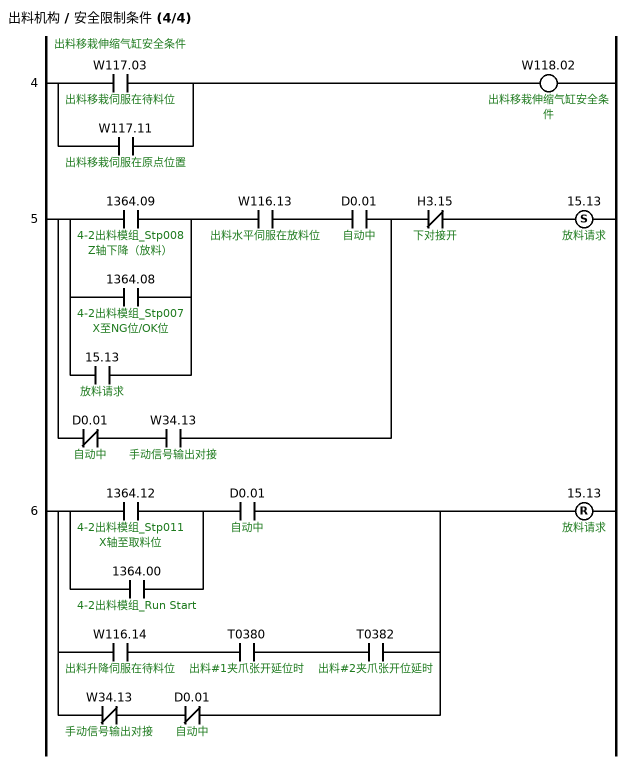
; [picture p336: 出料机构 / 安全限制条件, rungs 4-6]
; rung 4: 出料移栽伸缩气缸安全条件
LD W117.03  ; 出料移栽伺服在待料位
OR W117.11  ; 出料移栽伺服在原点位置
OUT W118.02  ; 出料移栽伸缩气缸安全条件
; rung 5
LD 1364.09  ; 4-2出料模组_Stp008 Z轴下降（放料）
OR 1364.08  ; 4-2出料模组_Stp007 X至NG位/OK位
OR 15.13  ; 放料请求
AND W116.13  ; 出料水平伺服在放料位
AND D0.01  ; 自动中
LDNOT D0.01  ; 自动中
AND W34.13  ; 手动信号输出对接
ORLD
ANDNOT H3.15  ; 下对接开
SET 15.13  ; 放料请求
; rung 6
LD 1364.12  ; 4-2出料模组_Stp011 X轴至取料位
OR 1364.00  ; 4-2出料模组_Run Start
AND D0.01  ; 自动中
LD W116.14  ; 出料升降伺服在待料位
AND T0380  ; 出料#1夹爪张开延位时
AND T0382  ; 出料#2夹爪张开位延时
ORLD
LDNOT W34.13  ; 手动信号输出对接
ANDNOT D0.01  ; 自动中
ORLD
RSET 15.13  ; 放料请求

### Section 出料机构输出

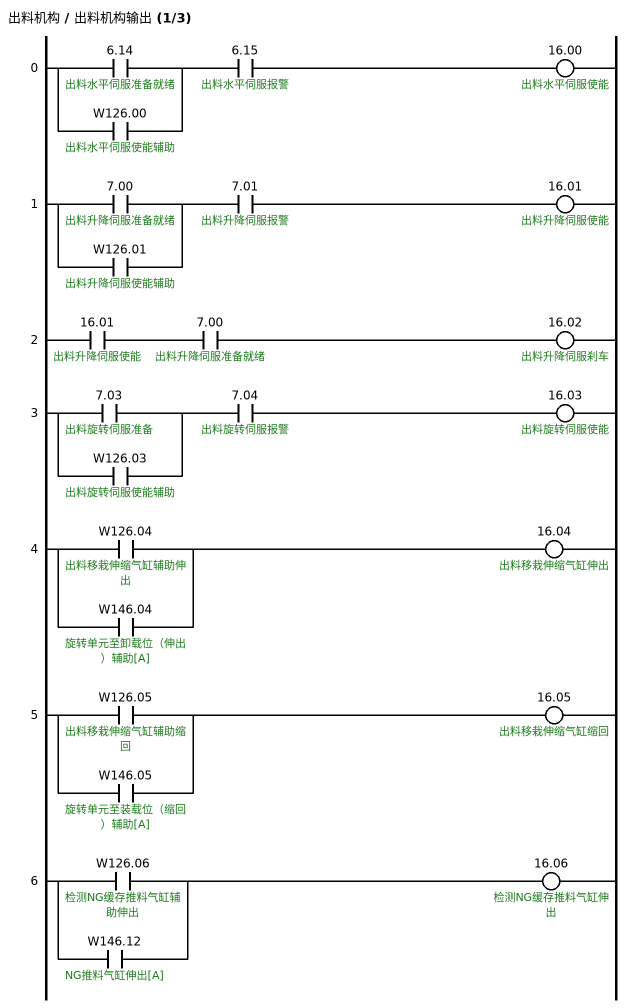
; rung 0
LD 6.14  ; 出料水平伺服准备就绪
OR W126.00  ; 出料水平伺服使能辅助
AND 6.15  ; 出料水平伺服报警
OUT 16.00  ; 出料水平伺服使能
; rung 1
LD 7.00  ; 出料升降伺服准备就绪
OR W126.01  ; 出料升降伺服使能辅助
AND 7.01  ; 出料升降伺服报警
OUT 16.01  ; 出料升降伺服使能
; rung 2
LD 16.01  ; 出料升降伺服使能
AND 7.00  ; 出料升降伺服准备就绪
OUT 16.02  ; 出料升降伺服刹车
; rung 3
LD 7.03  ; 出料旋转伺服准备
OR W126.03  ; 出料旋转伺服使能辅助
AND 7.04  ; 出料旋转伺服报警
OUT 16.03  ; 出料旋转伺服使能
; rung 4
LD W126.04  ; 出料移栽伸缩气缸辅助伸出
OR W146.04  ; 旋转单元至卸载位（伸出）辅助[A]
OUT 16.04  ; 出料移栽伸缩气缸伸出
; rung 5
LD W126.05  ; 出料移栽伸缩气缸辅助缩回
OR W146.05  ; 旋转单元至装载位（缩回）辅助[A]
OUT 16.05  ; 出料移栽伸缩气缸缩回
; rung 6
LD W126.06  ; 检测NG缓存推料气缸辅助伸出
OR W146.12  ; NG推料气缸伸出[A]
OUT 16.06  ; 检测NG缓存推料气缸伸出

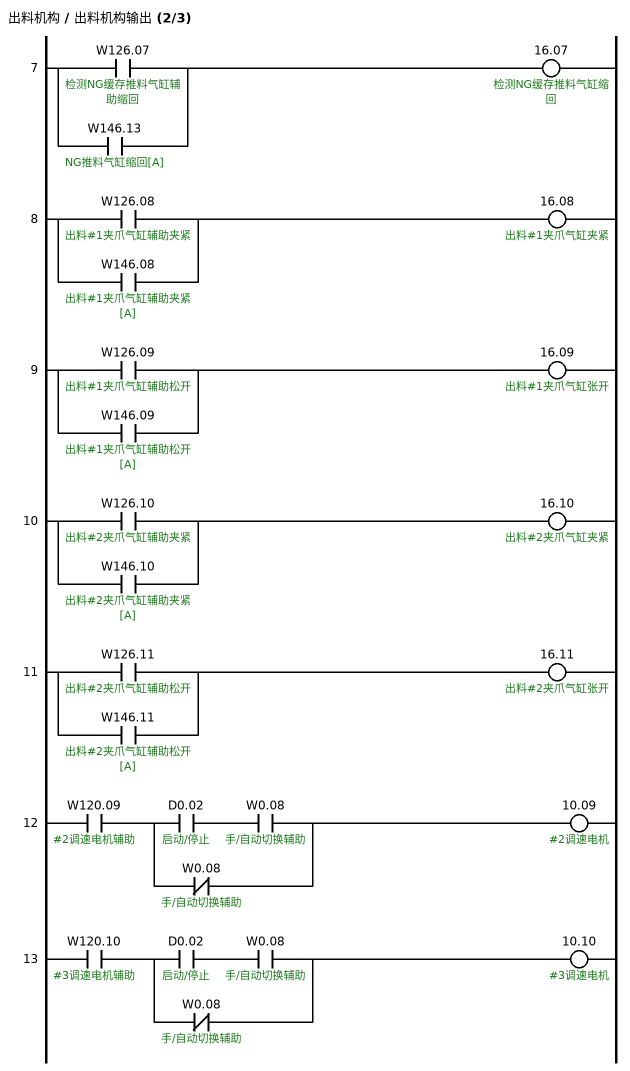
; rung 7
LD W126.07  ; 检测NG缓存推料气缸辅助缩回
OR W146.13  ; NG推料气缸缩回[A]
OUT 16.07  ; 检测NG缓存推料气缸缩回
; rung 8
LD W126.08  ; 出料#1夹爪气缸辅助夹紧
OR W146.08  ; 出料#1夹爪气缸辅助夹紧[A]
OUT 16.08  ; 出料#1夹爪气缸夹紧
; rung 9
LD W126.09  ; 出料#1夹爪气缸辅助松开
OR W146.09  ; 出料#1夹爪气缸辅助松开[A]
OUT 16.09  ; 出料#1夹爪气缸张开
; rung 10
LD W126.10  ; 出料#2夹爪气缸辅助夹紧
OR W146.10  ; 出料#2夹爪气缸辅助夹紧[A]
OUT 16.10  ; 出料#2夹爪气缸夹紧
; rung 11
LD W126.11  ; 出料#2夹爪气缸辅助松开
OR W146.11  ; 出料#2夹爪气缸辅助松开[A]
OUT 16.11  ; 出料#2夹爪气缸张开
; rung 12
LD W120.09  ; #2调速电机辅助
LD D0.02  ; 启动/停止
AND W0.08  ; 手/自动切换辅助
ORNOT W0.08  ; 手/自动切换辅助
ANDLD
OUT 10.09  ; #2调速电机
; rung 13
LD W120.10  ; #3调速电机辅助
LD D0.02  ; 启动/停止
AND W0.08  ; 手/自动切换辅助
ORNOT W0.08  ; 手/自动切换辅助
ANDLD
OUT 10.10  ; #3调速电机

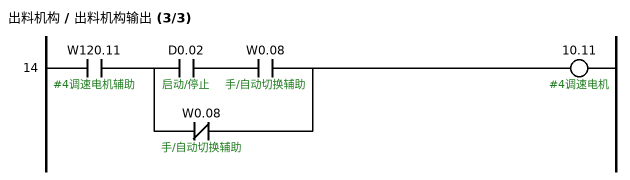
; rung 14
LD W120.11  ; #4调速电机辅助
LD D0.02  ; 启动/停止
AND W0.08  ; 手/自动切换辅助
ORNOT W0.08  ; 手/自动切换辅助
ANDLD
OUT 10.11  ; #4调速电机

### Section 出料机构手动

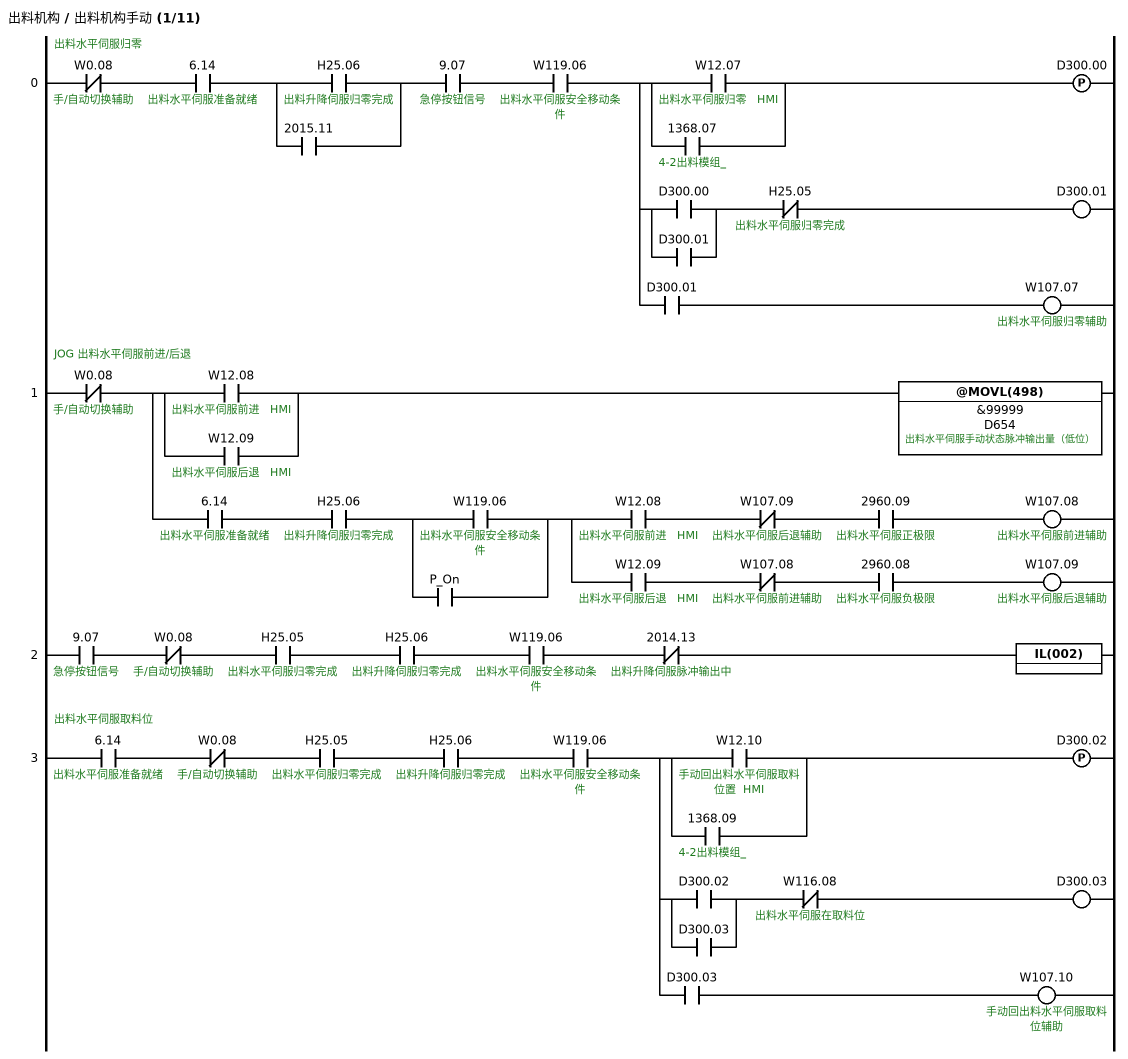
; rung 0: 出料水平伺服归零
LDNOT W0.08  ; 手/自动切换辅助
AND 6.14  ; 出料水平伺服准备就绪
LD H25.06  ; 出料升降伺服归零完成
OR 2015.11
ANDLD
AND 9.07  ; 急停按钮信号
AND W119.06  ; 出料水平伺服安全移动条件
OUT TR0
LD W12.07  ; 出料水平伺服归零   HMI
OR 1368.07  ; 4-2出料模组_
ANDLD
DIFU(013) D300.00
LD TR0
LD D300.00
OR D300.01
ANDLD
ANDNOT H25.05  ; 出料水平伺服归零完成
OUT D300.01
LD TR0
AND D300.01
OUT W107.07  ; 出料水平伺服归零辅助
; rung 1: JOG 出料水平伺服前进/后退
LDNOT W0.08  ; 手/自动切换辅助
OUT TR0
LD W12.08  ; 出料水平伺服前进   HMI
OR W12.09  ; 出料水平伺服后退   HMI
ANDLD
@MOVL(498) &99999 D654  ; 出料水平伺服手动状态脉冲输出量（低位）
LD TR0
AND 6.14  ; 出料水平伺服准备就绪
AND H25.06  ; 出料升降伺服归零完成
LD W119.06  ; 出料水平伺服安全移动条件
OR P_On
ANDLD
OUT TR0
AND W12.08  ; 出料水平伺服前进   HMI
ANDNOT W107.09  ; 出料水平伺服后退辅助
AND 2960.09  ; 出料水平伺服正极限
OUT W107.08  ; 出料水平伺服前进辅助
LD TR0
AND W12.09  ; 出料水平伺服后退   HMI
ANDNOT W107.08  ; 出料水平伺服前进辅助
AND 2960.08  ; 出料水平伺服负极限
OUT W107.09  ; 出料水平伺服后退辅助
; rung 2
LD 9.07  ; 急停按钮信号
ANDNOT W0.08  ; 手/自动切换辅助
AND H25.05  ; 出料水平伺服归零完成
AND H25.06  ; 出料升降伺服归零完成
AND W119.06  ; 出料水平伺服安全移动条件
ANDNOT 2014.13  ; 出料升降伺服脉冲输出中
IL(002)
; rung 3: 出料水平伺服取料位
LD 6.14  ; 出料水平伺服准备就绪
ANDNOT W0.08  ; 手/自动切换辅助
AND H25.05  ; 出料水平伺服归零完成
AND H25.06  ; 出料升降伺服归零完成
AND W119.06  ; 出料水平伺服安全移动条件
OUT TR0
LD W12.10  ; 手动回出料水平伺服取料位置  HMI
OR 1368.09  ; 4-2出料模组_
ANDLD
DIFU(013) D300.02
LD TR0
LD D300.02
OR D300.03
ANDLD
ANDNOT W116.08  ; 出料水平伺服在取料位
OUT D300.03
LD TR0
AND D300.03
OUT W107.10  ; 手动回出料水平伺服取料位辅助

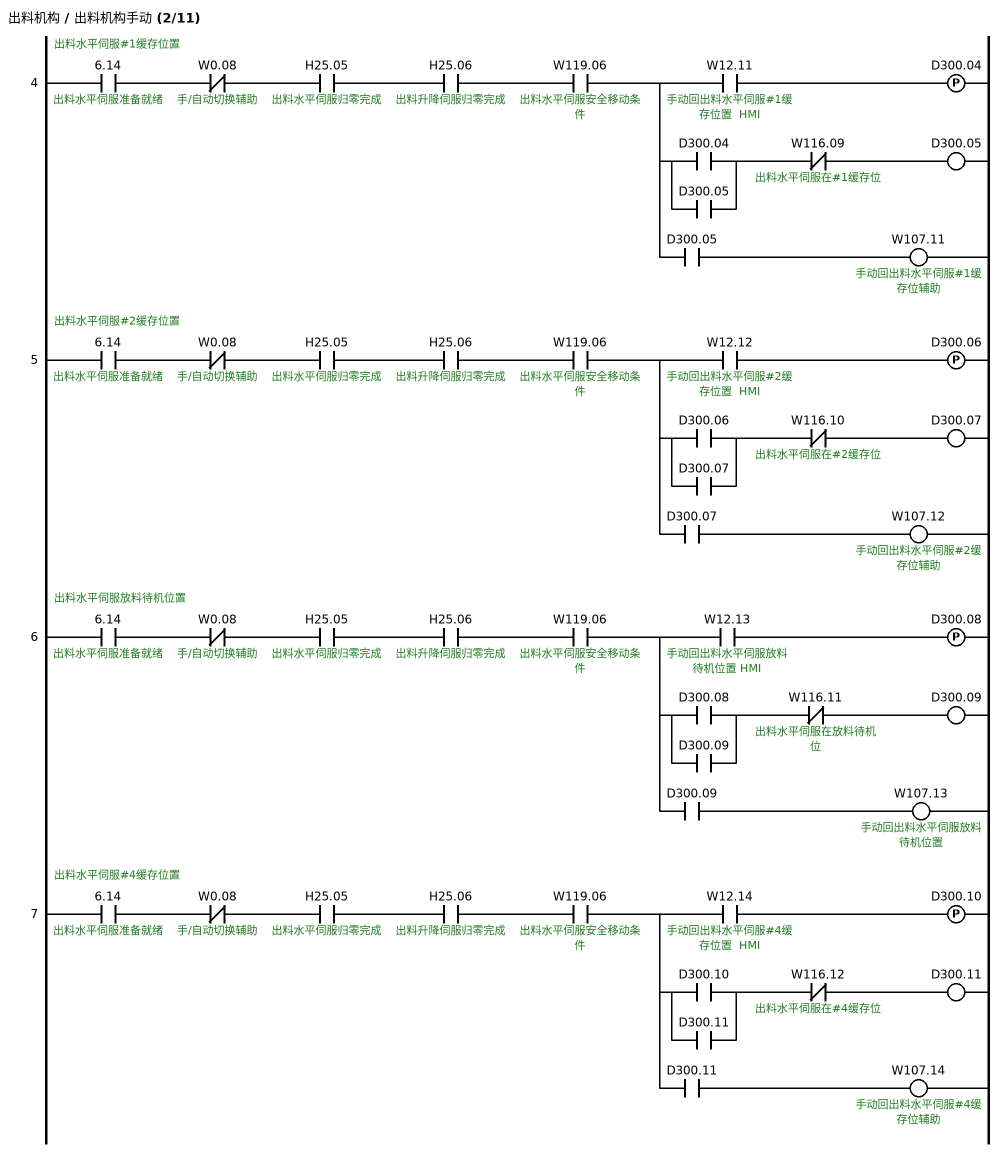
; rung 4: 出料水平伺服#1缓存位置
LD 6.14  ; 出料水平伺服准备就绪
ANDNOT W0.08  ; 手/自动切换辅助
AND H25.05  ; 出料水平伺服归零完成
AND H25.06  ; 出料升降伺服归零完成
AND W119.06  ; 出料水平伺服安全移动条件
OUT TR0
AND W12.11  ; 手动回出料水平伺服#1缓存位置  HMI
DIFU(013) D300.04
LD TR0
LD D300.04
OR D300.05
ANDLD
ANDNOT W116.09  ; 出料水平伺服在#1缓存位
OUT D300.05
LD TR0
AND D300.05
OUT W107.11  ; 手动回出料水平伺服#1缓存位辅助
; rung 5: 出料水平伺服#2缓存位置
LD 6.14  ; 出料水平伺服准备就绪
ANDNOT W0.08  ; 手/自动切换辅助
AND H25.05  ; 出料水平伺服归零完成
AND H25.06  ; 出料升降伺服归零完成
AND W119.06  ; 出料水平伺服安全移动条件
OUT TR0
AND W12.12  ; 手动回出料水平伺服#2缓存位置  HMI
DIFU(013) D300.06
LD TR0
LD D300.06
OR D300.07
ANDLD
ANDNOT W116.10  ; 出料水平伺服在#2缓存位
OUT D300.07
LD TR0
AND D300.07
OUT W107.12  ; 手动回出料水平伺服#2缓存位辅助
; rung 6: 出料水平伺服放料待机位置
LD 6.14  ; 出料水平伺服准备就绪
ANDNOT W0.08  ; 手/自动切换辅助
AND H25.05  ; 出料水平伺服归零完成
AND H25.06  ; 出料升降伺服归零完成
AND W119.06  ; 出料水平伺服安全移动条件
OUT TR0
AND W12.13  ; 手动回出料水平伺服放料待机位置 HMI
DIFU(013) D300.08
LD TR0
LD D300.08
OR D300.09
ANDLD
ANDNOT W116.11  ; 出料水平伺服在放料待机位
OUT D300.09
LD TR0
AND D300.09
OUT W107.13  ; 手动回出料水平伺服放料待机位置
; rung 7: 出料水平伺服#4缓存位置
LD 6.14  ; 出料水平伺服准备就绪
ANDNOT W0.08  ; 手/自动切换辅助
AND H25.05  ; 出料水平伺服归零完成
AND H25.06  ; 出料升降伺服归零完成
AND W119.06  ; 出料水平伺服安全移动条件
OUT TR0
AND W12.14  ; 手动回出料水平伺服#4缓存位置  HMI
DIFU(013) D300.10
LD TR0
LD D300.10
OR D300.11
ANDLD
ANDNOT W116.12  ; 出料水平伺服在#4缓存位
OUT D300.11
LD TR0
AND D300.11
OUT W107.14  ; 手动回出料水平伺服#4缓存位辅助

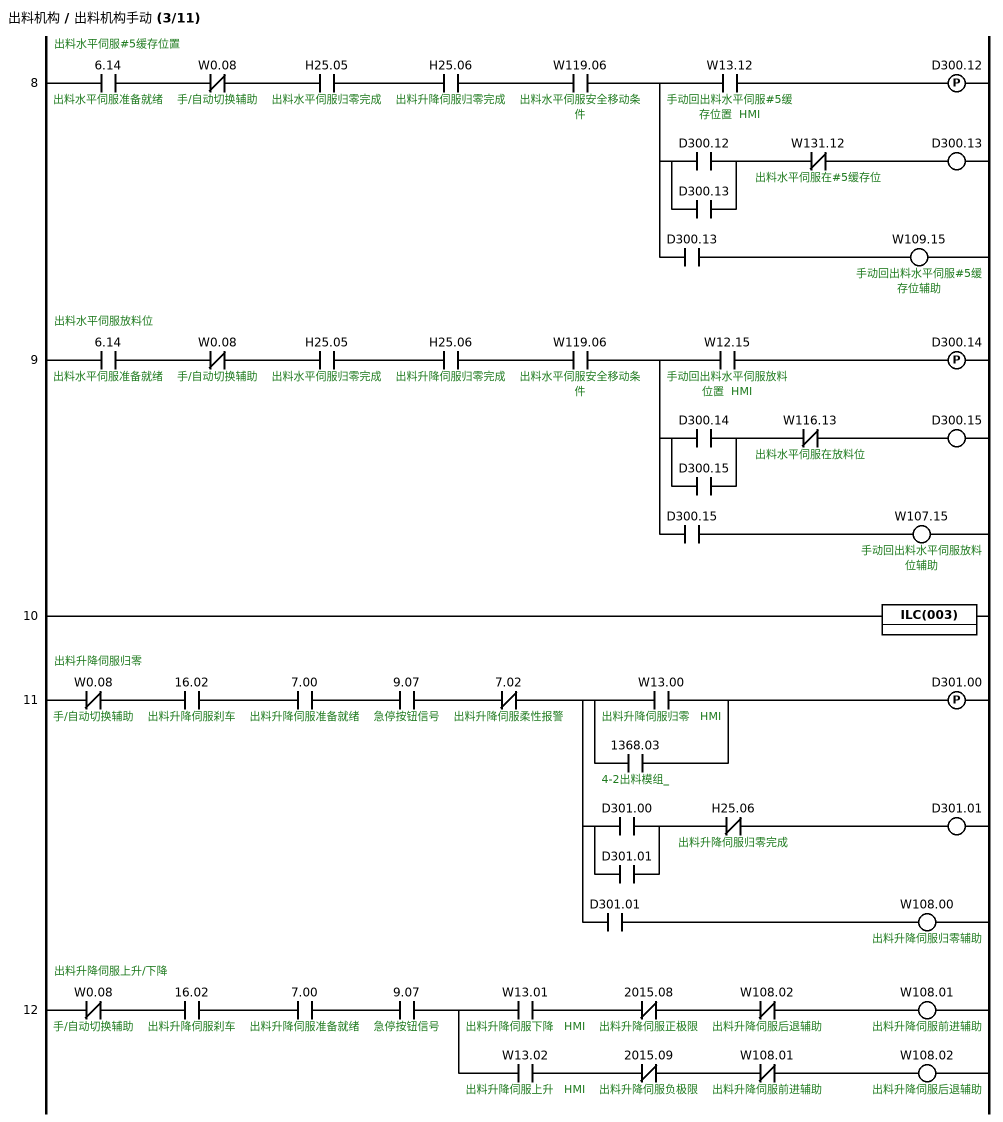
; rung 8: 出料水平伺服#5缓存位置
LD 6.14  ; 出料水平伺服准备就绪
ANDNOT W0.08  ; 手/自动切换辅助
AND H25.05  ; 出料水平伺服归零完成
AND H25.06  ; 出料升降伺服归零完成
AND W119.06  ; 出料水平伺服安全移动条件
OUT TR0
AND W13.12  ; 手动回出料水平伺服#5缓存位置  HMI
DIFU(013) D300.12
LD TR0
LD D300.12
OR D300.13
ANDLD
ANDNOT W131.12  ; 出料水平伺服在#5缓存位
OUT D300.13
LD TR0
AND D300.13
OUT W109.15  ; 手动回出料水平伺服#5缓存位辅助
; rung 9: 出料水平伺服放料位
LD 6.14  ; 出料水平伺服准备就绪
ANDNOT W0.08  ; 手/自动切换辅助
AND H25.05  ; 出料水平伺服归零完成
AND H25.06  ; 出料升降伺服归零完成
AND W119.06  ; 出料水平伺服安全移动条件
OUT TR0
AND W12.15  ; 手动回出料水平伺服放料位置  HMI
DIFU(013) D300.14
LD TR0
LD D300.14
OR D300.15
ANDLD
ANDNOT W116.13  ; 出料水平伺服在放料位
OUT D300.15
LD TR0
AND D300.15
OUT W107.15  ; 手动回出料水平伺服放料位辅助
; rung 10
ILC(003)
; rung 11: 出料升降伺服归零
LDNOT W0.08  ; 手/自动切换辅助
AND 16.02  ; 出料升降伺服刹车
AND 7.00  ; 出料升降伺服准备就绪
AND 9.07  ; 急停按钮信号
ANDNOT 7.02  ; 出料升降伺服柔性报警
OUT TR0
LD W13.00  ; 出料升降伺服归零   HMI
OR 1368.03  ; 4-2出料模组_
ANDLD
DIFU(013) D301.00
LD TR0
LD D301.00
OR D301.01
ANDLD
ANDNOT H25.06  ; 出料升降伺服归零完成
OUT D301.01
LD TR0
AND D301.01
OUT W108.00  ; 出料升降伺服归零辅助
; rung 12: 出料升降伺服上升/下降
LDNOT W0.08  ; 手/自动切换辅助
AND 16.02  ; 出料升降伺服刹车
AND 7.00  ; 出料升降伺服准备就绪
AND 9.07  ; 急停按钮信号
OUT TR0
AND W13.01  ; 出料升降伺服下降   HMI
ANDNOT 2015.08  ; 出料升降伺服正极限
ANDNOT W108.02  ; 出料升降伺服后退辅助
OUT W108.01  ; 出料升降伺服前进辅助
LD TR0
AND W13.02  ; 出料升降伺服上升   HMI
ANDNOT 2015.09  ; 出料升降伺服负极限
ANDNOT W108.01  ; 出料升降伺服前进辅助
OUT W108.02  ; 出料升降伺服后退辅助

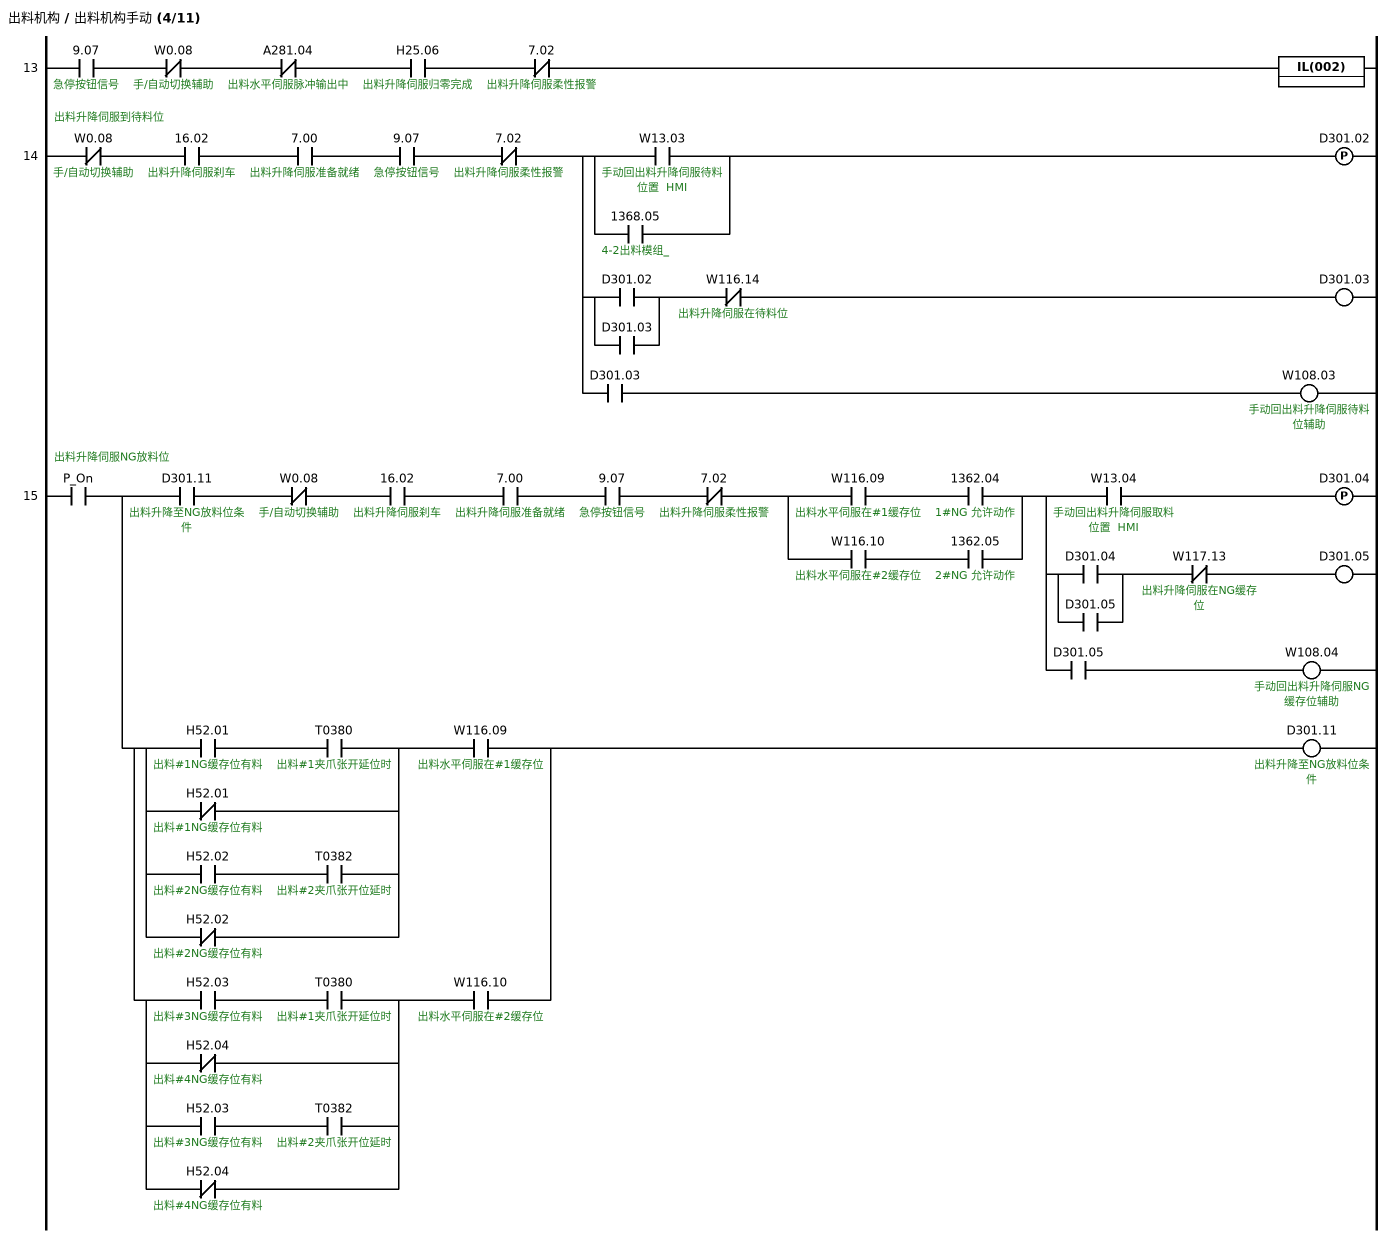
; rung 13
LD 9.07  ; 急停按钮信号
ANDNOT W0.08  ; 手/自动切换辅助
ANDNOT A281.04  ; 出料水平伺服脉冲输出中
AND H25.06  ; 出料升降伺服归零完成
ANDNOT 7.02  ; 出料升降伺服柔性报警
IL(002)
; rung 14: 出料升降伺服到待料位
LDNOT W0.08  ; 手/自动切换辅助
AND 16.02  ; 出料升降伺服刹车
AND 7.00  ; 出料升降伺服准备就绪
AND 9.07  ; 急停按钮信号
ANDNOT 7.02  ; 出料升降伺服柔性报警
OUT TR0
LD W13.03  ; 手动回出料升降伺服待料位置  HMI
OR 1368.05  ; 4-2出料模组_
ANDLD
DIFU(013) D301.02
LD TR0
LD D301.02
OR D301.03
ANDLD
ANDNOT W116.14  ; 出料升降伺服在待料位
OUT D301.03
LD TR0
AND D301.03
OUT W108.03  ; 手动回出料升降伺服待料位辅助
; rung 15: 出料升降伺服NG放料位
LD P_On
OUT TR0
AND D301.11  ; 出料升降至NG放料位条件
ANDNOT W0.08  ; 手/自动切换辅助
AND 16.02  ; 出料升降伺服刹车
AND 7.00  ; 出料升降伺服准备就绪
AND 9.07  ; 急停按钮信号
ANDNOT 7.02  ; 出料升降伺服柔性报警
LD W116.09  ; 出料水平伺服在#1缓存位
AND 1362.04  ; 1#NG 允许动作
LD W116.10  ; 出料水平伺服在#2缓存位
AND 1362.05  ; 2#NG 允许动作
ORLD
ANDLD
OUT TR1
AND W13.04  ; 手动回出料升降伺服取料位置  HMI
DIFU(013) D301.04
LD TR1
LD D301.04
OR D301.05
ANDLD
ANDNOT W117.13  ; 出料升降伺服在NG缓存位
OUT D301.05
LD TR1
AND D301.05
OUT W108.04  ; 手动回出料升降伺服NG缓存位辅助
LD TR0
LD H52.01  ; 出料#1NG缓存位有料
AND T0380  ; 出料#1夹爪张开延位时
ORNOT H52.01  ; 出料#1NG缓存位有料
LD H52.02  ; 出料#2NG缓存位有料
AND T0382  ; 出料#2夹爪张开位延时
ORLD
ORNOT H52.02  ; 出料#2NG缓存位有料
AND W116.09  ; 出料水平伺服在#1缓存位
LD H52.03  ; 出料#3NG缓存位有料
AND T0380  ; 出料#1夹爪张开延位时
ORNOT H52.04  ; 出料#4NG缓存位有料
LD H52.03  ; 出料#3NG缓存位有料
AND T0382  ; 出料#2夹爪张开位延时
ORLD
ORNOT H52.04  ; 出料#4NG缓存位有料
AND W116.10  ; 出料水平伺服在#2缓存位
ORLD
ANDLD
OUT D301.11  ; 出料升降至NG放料位条件

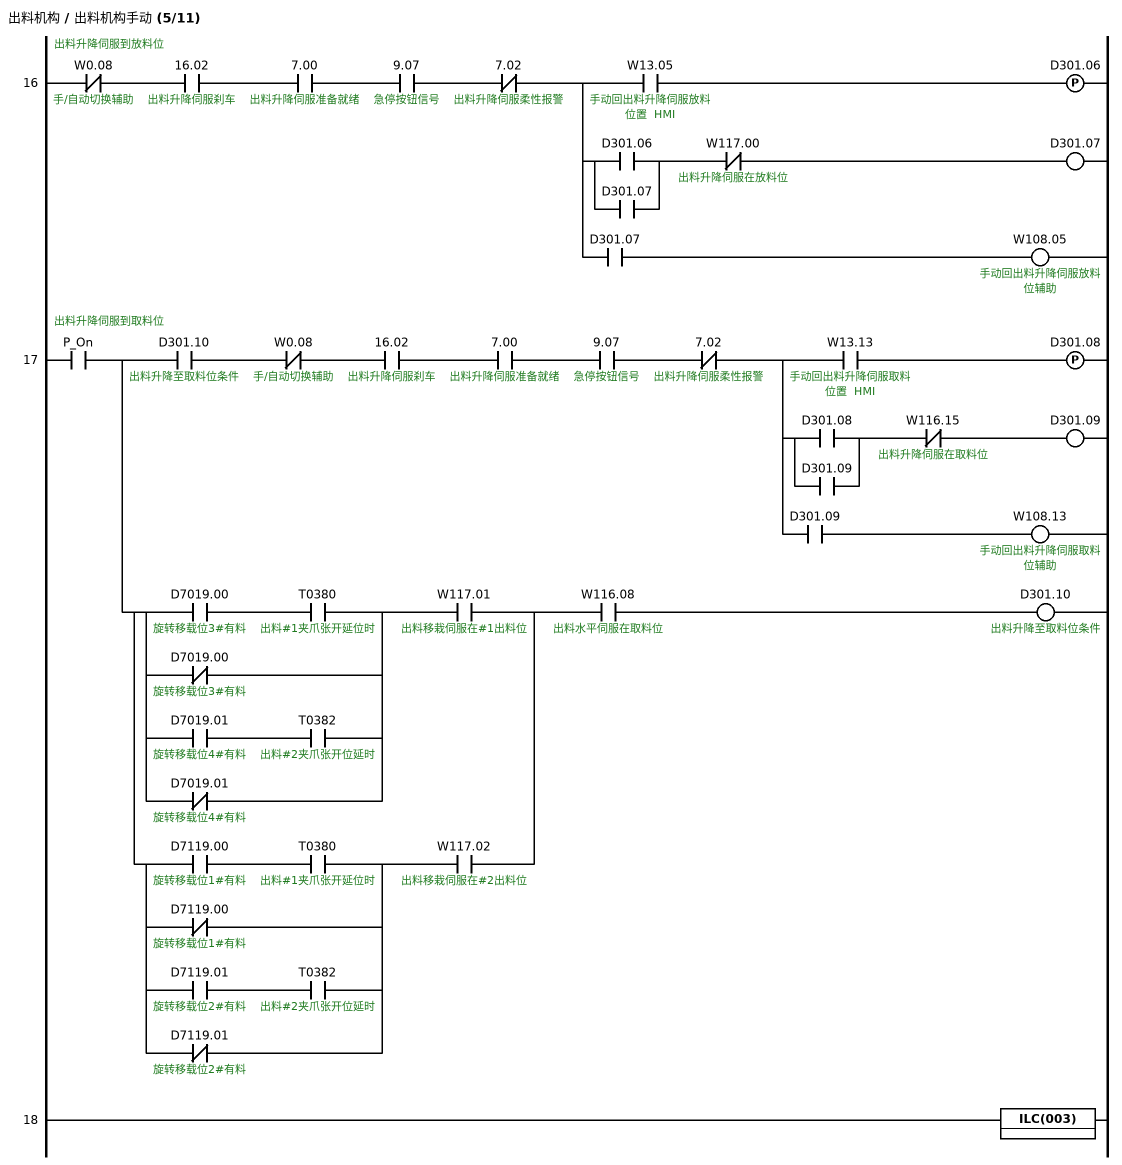
; rung 16: 出料升降伺服到放料位
LDNOT W0.08  ; 手/自动切换辅助
AND 16.02  ; 出料升降伺服刹车
AND 7.00  ; 出料升降伺服准备就绪
AND 9.07  ; 急停按钮信号
ANDNOT 7.02  ; 出料升降伺服柔性报警
OUT TR0
AND W13.05  ; 手动回出料升降伺服放料位置  HMI
DIFU(013) D301.06
LD TR0
LD D301.06
OR D301.07
ANDLD
ANDNOT W117.00  ; 出料升降伺服在放料位
OUT D301.07
LD TR0
AND D301.07
OUT W108.05  ; 手动回出料升降伺服放料位辅助
; rung 17: 出料升降伺服到取料位
LD P_On
OUT TR0
AND D301.10  ; 出料升降至取料位条件
ANDNOT W0.08  ; 手/自动切换辅助
AND 16.02  ; 出料升降伺服刹车
AND 7.00  ; 出料升降伺服准备就绪
AND 9.07  ; 急停按钮信号
ANDNOT 7.02  ; 出料升降伺服柔性报警
OUT TR1
AND W13.13  ; 手动回出料升降伺服取料位置  HMI
DIFU(013) D301.08
LD TR1
LD D301.08
OR D301.09
ANDLD
ANDNOT W116.15  ; 出料升降伺服在取料位
OUT D301.09
LD TR1
AND D301.09
OUT W108.13  ; 手动回出料升降伺服取料位辅助
LD TR0
LD D7019.00  ; 旋转移载位3#有料
AND T0380  ; 出料#1夹爪张开延位时
ORNOT D7019.00  ; 旋转移载位3#有料
LD D7019.01  ; 旋转移载位4#有料
AND T0382  ; 出料#2夹爪张开位延时
ORLD
ORNOT D7019.01  ; 旋转移载位4#有料
AND W117.01  ; 出料移栽伺服在#1出料位
LD D7119.00  ; 旋转移载位1#有料
AND T0380  ; 出料#1夹爪张开延位时
ORNOT D7119.00  ; 旋转移载位1#有料
LD D7119.01  ; 旋转移载位2#有料
AND T0382  ; 出料#2夹爪张开位延时
ORLD
ORNOT D7119.01  ; 旋转移载位2#有料
AND W117.02  ; 出料移栽伺服在#2出料位
ORLD
ANDLD
AND W116.08  ; 出料水平伺服在取料位
OUT D301.10  ; 出料升降至取料位条件
; rung 18
ILC(003)

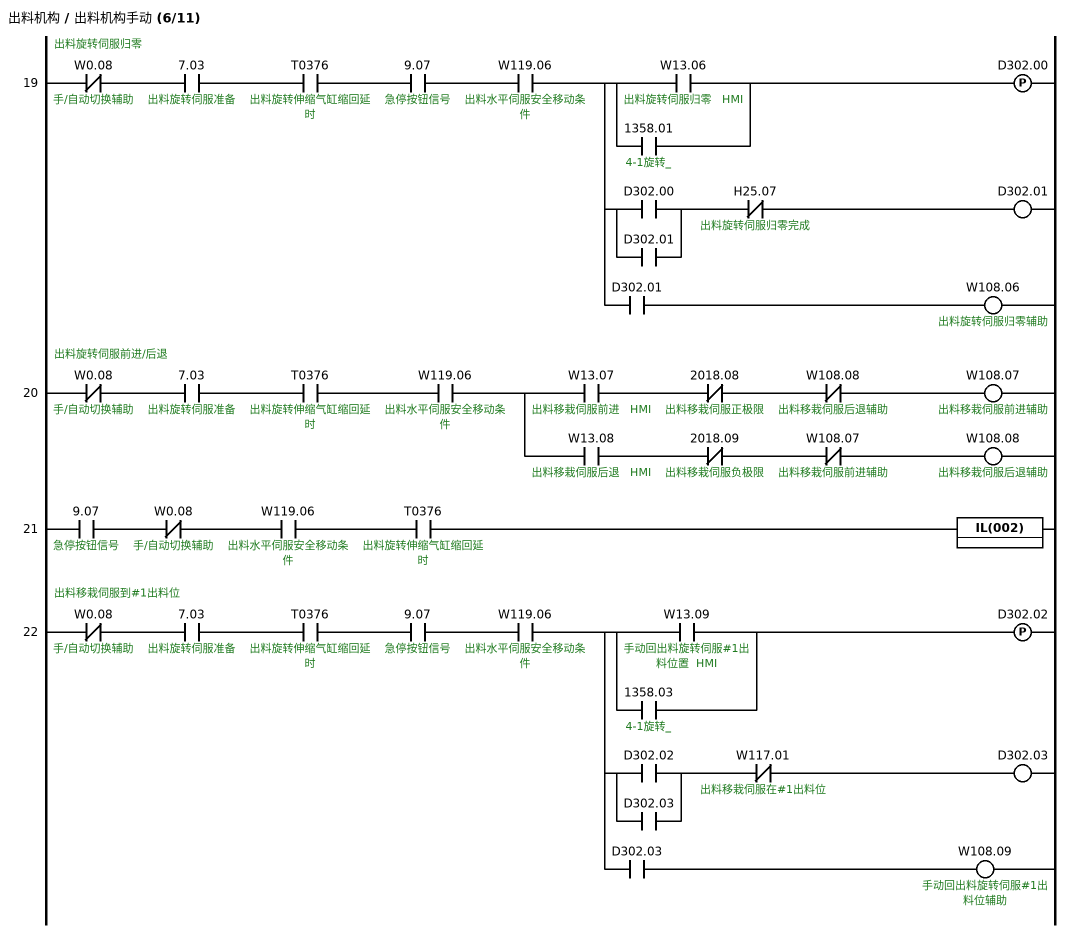
; rung 19: 出料旋转伺服归零
LDNOT W0.08  ; 手/自动切换辅助
AND 7.03  ; 出料旋转伺服准备
AND T0376  ; 出料旋转伸缩气缸缩回延时
AND 9.07  ; 急停按钮信号
AND W119.06  ; 出料水平伺服安全移动条件
OUT TR0
LD W13.06  ; 出料旋转伺服归零   HMI
OR 1358.01  ; 4-1旋转_
ANDLD
DIFU(013) D302.00
LD TR0
LD D302.00
OR D302.01
ANDLD
ANDNOT H25.07  ; 出料旋转伺服归零完成
OUT D302.01
LD TR0
AND D302.01
OUT W108.06  ; 出料旋转伺服归零辅助
; rung 20: 出料旋转伺服前进/后退
LDNOT W0.08  ; 手/自动切换辅助
AND 7.03  ; 出料旋转伺服准备
AND T0376  ; 出料旋转伸缩气缸缩回延时
AND W119.06  ; 出料水平伺服安全移动条件
OUT TR0
AND W13.07  ; 出料移栽伺服前进   HMI
ANDNOT 2018.08  ; 出料移栽伺服正极限
ANDNOT W108.08  ; 出料移栽伺服后退辅助
OUT W108.07  ; 出料移栽伺服前进辅助
LD TR0
AND W13.08  ; 出料移栽伺服后退   HMI
ANDNOT 2018.09  ; 出料移栽伺服负极限
ANDNOT W108.07  ; 出料移栽伺服前进辅助
OUT W108.08  ; 出料移栽伺服后退辅助
; rung 21
LD 9.07  ; 急停按钮信号
ANDNOT W0.08  ; 手/自动切换辅助
AND W119.06  ; 出料水平伺服安全移动条件
AND T0376  ; 出料旋转伸缩气缸缩回延时
IL(002)
; rung 22: 出料移栽伺服到#1出料位
LDNOT W0.08  ; 手/自动切换辅助
AND 7.03  ; 出料旋转伺服准备
AND T0376  ; 出料旋转伸缩气缸缩回延时
AND 9.07  ; 急停按钮信号
AND W119.06  ; 出料水平伺服安全移动条件
OUT TR0
LD W13.09  ; 手动回出料旋转伺服#1出料位置  HMI
OR 1358.03  ; 4-1旋转_
ANDLD
DIFU(013) D302.02
LD TR0
LD D302.02
OR D302.03
ANDLD
ANDNOT W117.01  ; 出料移栽伺服在#1出料位
OUT D302.03
LD TR0
AND D302.03
OUT W108.09  ; 手动回出料旋转伺服#1出料位辅助

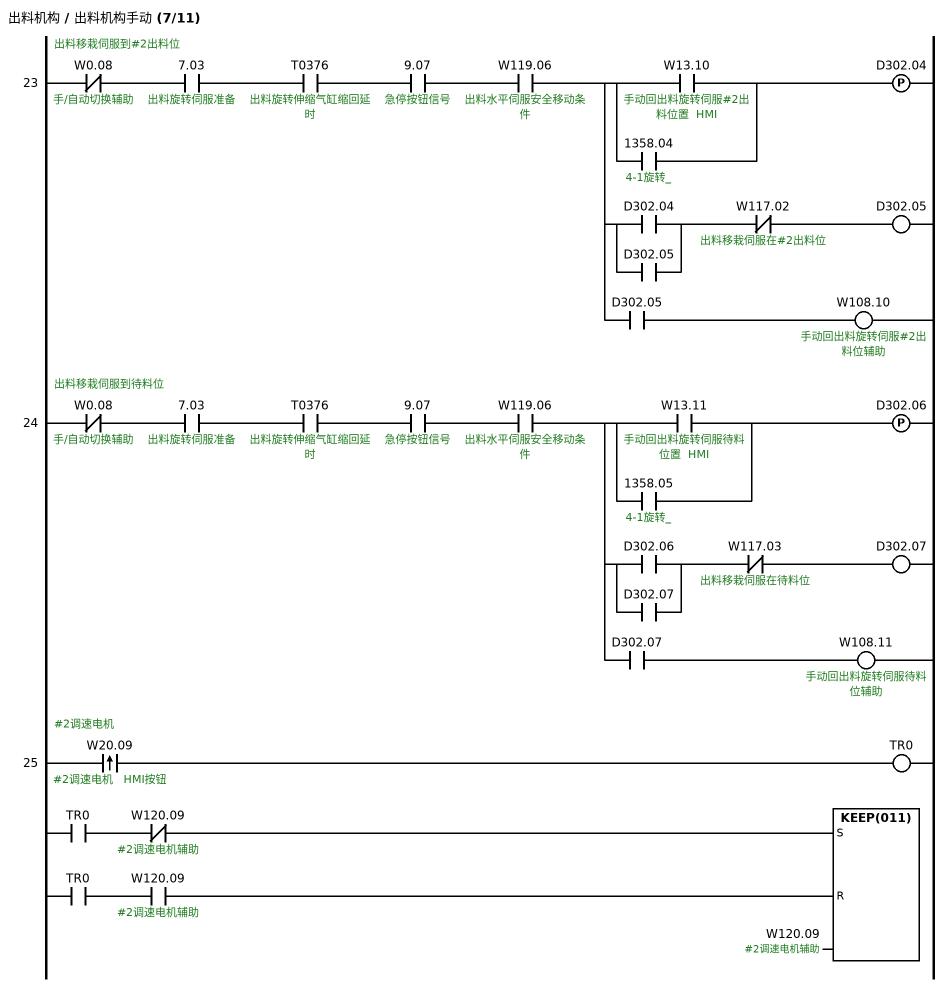
; rung 23: 出料移栽伺服到#2出料位
LDNOT W0.08  ; 手/自动切换辅助
AND 7.03  ; 出料旋转伺服准备
AND T0376  ; 出料旋转伸缩气缸缩回延时
AND 9.07  ; 急停按钮信号
AND W119.06  ; 出料水平伺服安全移动条件
OUT TR0
LD W13.10  ; 手动回出料旋转伺服#2出料位置  HMI
OR 1358.04  ; 4-1旋转_
ANDLD
DIFU(013) D302.04
LD TR0
LD D302.04
OR D302.05
ANDLD
ANDNOT W117.02  ; 出料移栽伺服在#2出料位
OUT D302.05
LD TR0
AND D302.05
OUT W108.10  ; 手动回出料旋转伺服#2出料位辅助
; rung 24: 出料移栽伺服到待料位
LDNOT W0.08  ; 手/自动切换辅助
AND 7.03  ; 出料旋转伺服准备
AND T0376  ; 出料旋转伸缩气缸缩回延时
AND 9.07  ; 急停按钮信号
AND W119.06  ; 出料水平伺服安全移动条件
OUT TR0
LD W13.11  ; 手动回出料旋转伺服待料位置  HMI
OR 1358.05  ; 4-1旋转_
ANDLD
DIFU(013) D302.06
LD TR0
LD D302.06
OR D302.07
ANDLD
ANDNOT W117.03  ; 出料移栽伺服在待料位
OUT D302.07
LD TR0
AND D302.07
OUT W108.11  ; 手动回出料旋转伺服待料位辅助
; rung 25: #2调速电机
@LD W20.09  ; #2调速电机   HMI按钮
OUT TR0
ANDNOT W120.09  ; #2调速电机辅助
LD TR0
AND W120.09  ; #2调速电机辅助
KEEP(011) W120.09  ; #2调速电机辅助

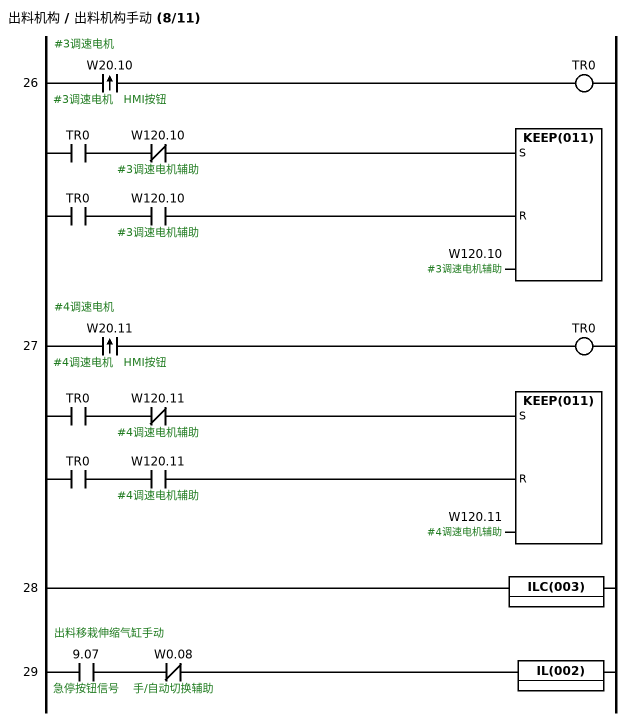
; rung 26: #3调速电机
@LD W20.10  ; #3调速电机   HMI按钮
OUT TR0
ANDNOT W120.10  ; #3调速电机辅助
LD TR0
AND W120.10  ; #3调速电机辅助
KEEP(011) W120.10  ; #3调速电机辅助
; rung 27: #4调速电机
@LD W20.11  ; #4调速电机   HMI按钮
OUT TR0
ANDNOT W120.11  ; #4调速电机辅助
LD TR0
AND W120.11  ; #4调速电机辅助
KEEP(011) W120.11  ; #4调速电机辅助
; rung 28
ILC(003)
; rung 29: 出料移栽伸缩气缸手动
LD 9.07  ; 急停按钮信号
ANDNOT W0.08  ; 手/自动切换辅助
IL(002)

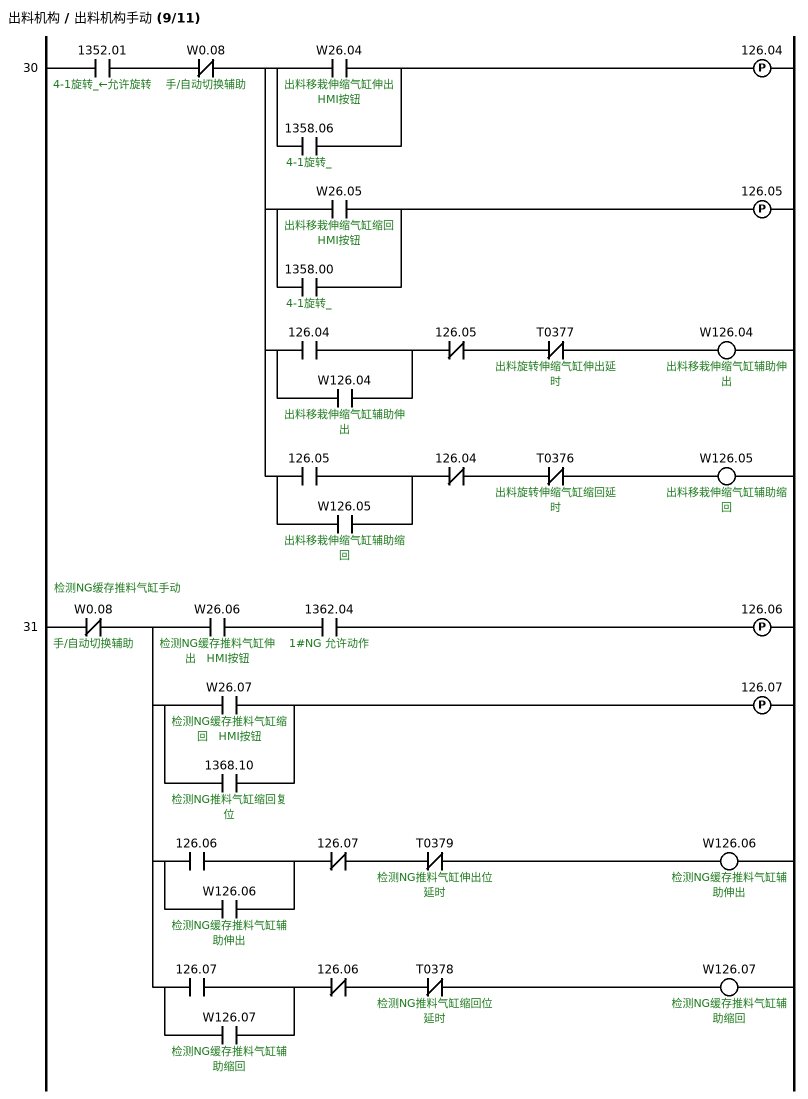
; rung 30
LD 1352.01  ; 4-1旋转_←允许旋转
ANDNOT W0.08  ; 手/自动切换辅助
OUT TR0
LD W26.04  ; 出料移栽伸缩气缸伸出  HMI按钮
OR 1358.06  ; 4-1旋转_
ANDLD
DIFU(013) 126.04
LD TR0
LD W26.05  ; 出料移栽伸缩气缸缩回  HMI按钮
OR 1358.00  ; 4-1旋转_
ANDLD
DIFU(013) 126.05
LD TR0
LD 126.04
OR W126.04  ; 出料移栽伸缩气缸辅助伸出
ANDLD
ANDNOT 126.05
ANDNOT T0377  ; 出料旋转伸缩气缸伸出延时
OUT W126.04  ; 出料移栽伸缩气缸辅助伸出
LD TR0
LD 126.05
OR W126.05  ; 出料移栽伸缩气缸辅助缩回
ANDLD
ANDNOT 126.04
ANDNOT T0376  ; 出料旋转伸缩气缸缩回延时
OUT W126.05  ; 出料移栽伸缩气缸辅助缩回
; rung 31: 检测NG缓存推料气缸手动
LDNOT W0.08  ; 手/自动切换辅助
OUT TR0
AND W26.06  ; 检测NG缓存推料气缸伸出   HMI按钮
AND 1362.04  ; 1#NG 允许动作
DIFU(013) 126.06
LD TR0
LD W26.07  ; 检测NG缓存推料气缸缩回   HMI按钮
OR 1368.10  ; 检测NG推料气缸缩回复位
ANDLD
DIFU(013) 126.07
LD TR0
LD 126.06
OR W126.06  ; 检测NG缓存推料气缸辅助伸出
ANDLD
ANDNOT 126.07
ANDNOT T0379  ; 检测NG推料气缸伸出位延时
OUT W126.06  ; 检测NG缓存推料气缸辅助伸出
LD TR0
LD 126.07
OR W126.07  ; 检测NG缓存推料气缸辅助缩回
ANDLD
ANDNOT 126.06
ANDNOT T0378  ; 检测NG推料气缸缩回位延时
OUT W126.07  ; 检测NG缓存推料气缸辅助缩回

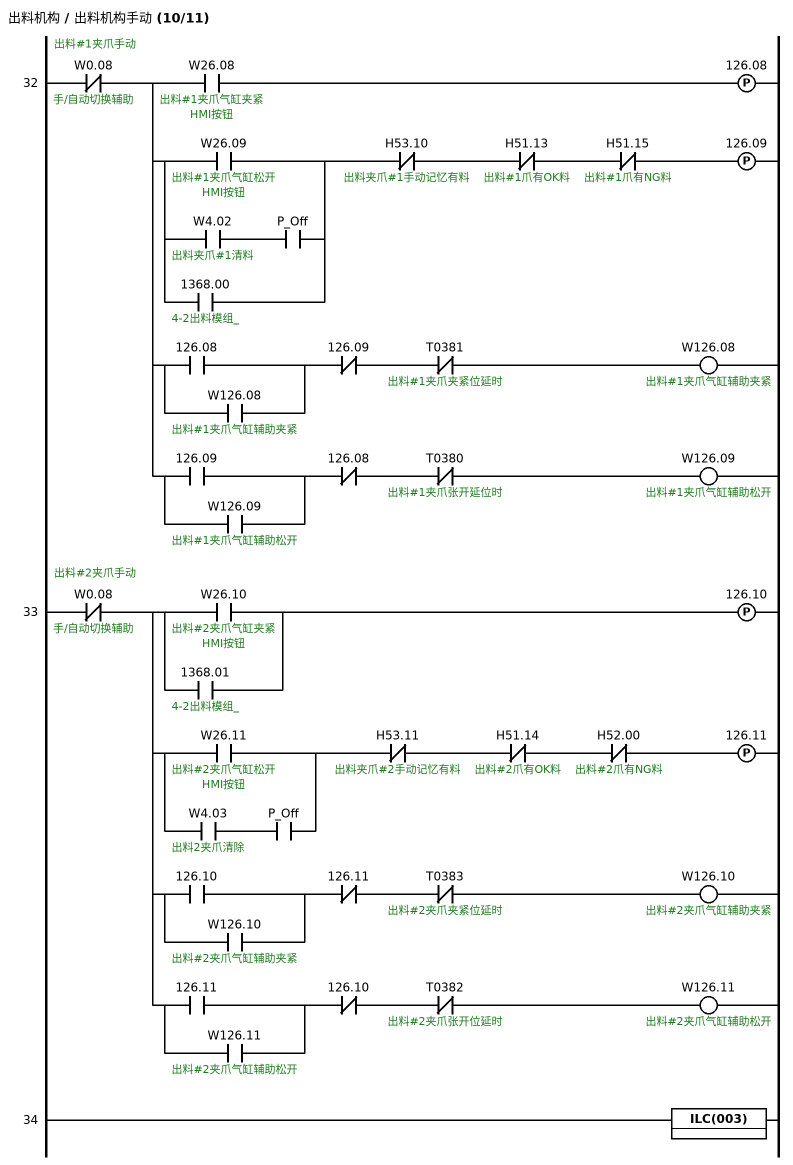
; rung 32: 出料#1夹爪手动
LDNOT W0.08  ; 手/自动切换辅助
OUT TR0
AND W26.08  ; 出料#1夹爪气缸夹紧   HMI按钮
DIFU(013) 126.08
LD TR0
LD W26.09  ; 出料#1夹爪气缸松开   HMI按钮
LD W4.02  ; 出料夹爪#1清料
AND P_Off
ORLD
OR 1368.00  ; 4-2出料模组_
ANDLD
ANDNOT H53.10  ; 出料夹爪#1手动记忆有料
ANDNOT H51.13  ; 出料#1爪有OK料
ANDNOT H51.15  ; 出料#1爪有NG料
DIFU(013) 126.09
LD TR0
LD 126.08
OR W126.08  ; 出料#1夹爪气缸辅助夹紧
ANDLD
ANDNOT 126.09
ANDNOT T0381  ; 出料#1夹爪夹紧位延时
OUT W126.08  ; 出料#1夹爪气缸辅助夹紧
LD TR0
LD 126.09
OR W126.09  ; 出料#1夹爪气缸辅助松开
ANDLD
ANDNOT 126.08
ANDNOT T0380  ; 出料#1夹爪张开延位时
OUT W126.09  ; 出料#1夹爪气缸辅助松开
; rung 33: 出料#2夹爪手动
LDNOT W0.08  ; 手/自动切换辅助
OUT TR0
LD W26.10  ; 出料#2夹爪气缸夹紧   HMI按钮
OR 1368.01  ; 4-2出料模组_
ANDLD
DIFU(013) 126.10
LD TR0
LD W26.11  ; 出料#2夹爪气缸松开   HMI按钮
LD W4.03  ; 出料2夹爪清除
AND P_Off
ORLD
ANDLD
ANDNOT H53.11  ; 出料夹爪#2手动记忆有料
ANDNOT H51.14  ; 出料#2爪有OK料
ANDNOT H52.00  ; 出料#2爪有NG料
DIFU(013) 126.11
LD TR0
LD 126.10
OR W126.10  ; 出料#2夹爪气缸辅助夹紧
ANDLD
ANDNOT 126.11
ANDNOT T0383  ; 出料#2夹爪夹紧位延时
OUT W126.10  ; 出料#2夹爪气缸辅助夹紧
LD TR0
LD 126.11
OR W126.11  ; 出料#2夹爪气缸辅助松开
ANDLD
ANDNOT 126.10
ANDNOT T0382  ; 出料#2夹爪张开位延时
OUT W126.11  ; 出料#2夹爪气缸辅助松开
; rung 34
ILC(003)

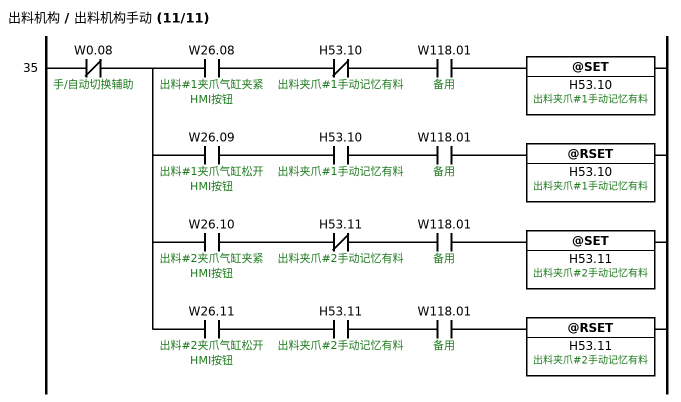
; rung 35
LDNOT W0.08  ; 手/自动切换辅助
OUT TR0
AND W26.08  ; 出料#1夹爪气缸夹紧   HMI按钮
ANDNOT H53.10  ; 出料夹爪#1手动记忆有料
AND W118.01  ; 备用
@SET H53.10  ; 出料夹爪#1手动记忆有料
LD TR0
AND W26.09  ; 出料#1夹爪气缸松开   HMI按钮
AND H53.10  ; 出料夹爪#1手动记忆有料
AND W118.01  ; 备用
@RSET H53.10  ; 出料夹爪#1手动记忆有料
LD TR0
AND W26.10  ; 出料#2夹爪气缸夹紧   HMI按钮
ANDNOT H53.11  ; 出料夹爪#2手动记忆有料
AND W118.01  ; 备用
@SET H53.11  ; 出料夹爪#2手动记忆有料
LD TR0
AND W26.11  ; 出料#2夹爪气缸松开   HMI按钮
AND H53.11  ; 出料夹爪#2手动记忆有料
AND W118.01  ; 备用
@RSET H53.11  ; 出料夹爪#2手动记忆有料

### Section 出料水平伺服参数设置

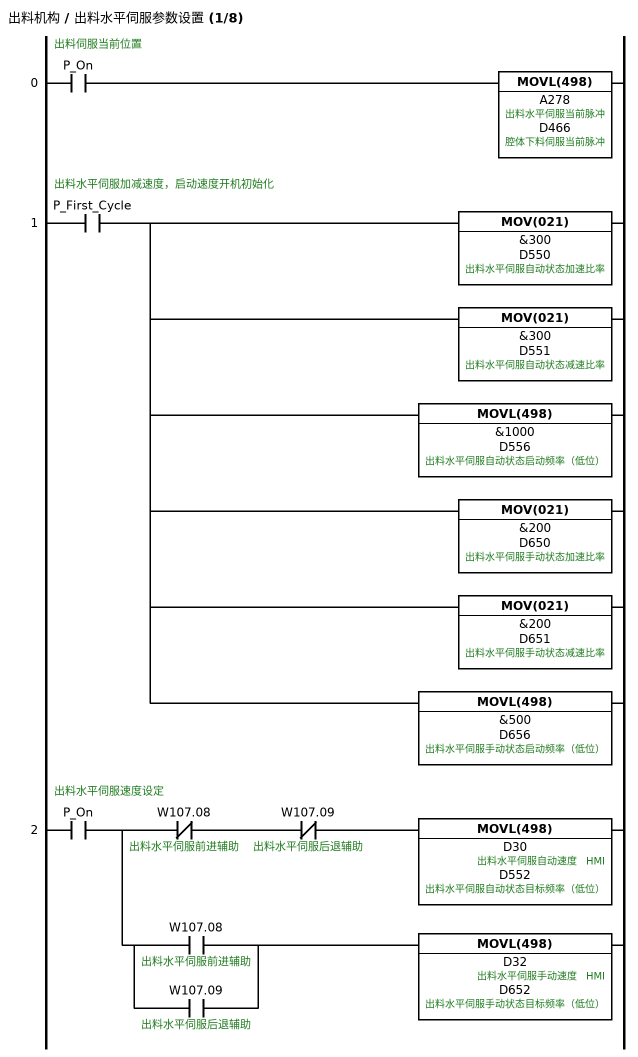
; rung 0: 出料伺服当前位置
LD P_On
MOVL(498) A278 D466  ; 出料水平伺服当前脉冲, 腔体下料伺服当前脉冲
; rung 1: 出料水平伺服加减速度，启动速度开机初始化
LD P_First_Cycle
MOV(021) &300 D550  ; 出料水平伺服自动状态加速比率
MOV(021) &300 D551  ; 出料水平伺服自动状态减速比率
MOVL(498) &1000 D556  ; 出料水平伺服自动状态启动频率（低位）
MOV(021) &200 D650  ; 出料水平伺服手动状态加速比率
MOV(021) &200 D651  ; 出料水平伺服手动状态减速比率
MOVL(498) &500 D656  ; 出料水平伺服手动状态启动频率（低位）
; rung 2: 出料水平伺服速度设定
LD P_On
OUT TR0
ANDNOT W107.08  ; 出料水平伺服前进辅助
ANDNOT W107.09  ; 出料水平伺服后退辅助
MOVL(498) D30 D552  ; 出料水平伺服自动速度   HMI, 出料水平伺服自动状态目标频率（低位）
LD TR0
LD W107.08  ; 出料水平伺服前进辅助
OR W107.09  ; 出料水平伺服后退辅助
ANDLD
MOVL(498) D32 D652  ; 出料水平伺服手动速度   HMI, 出料水平伺服手动状态目标频率（低位）

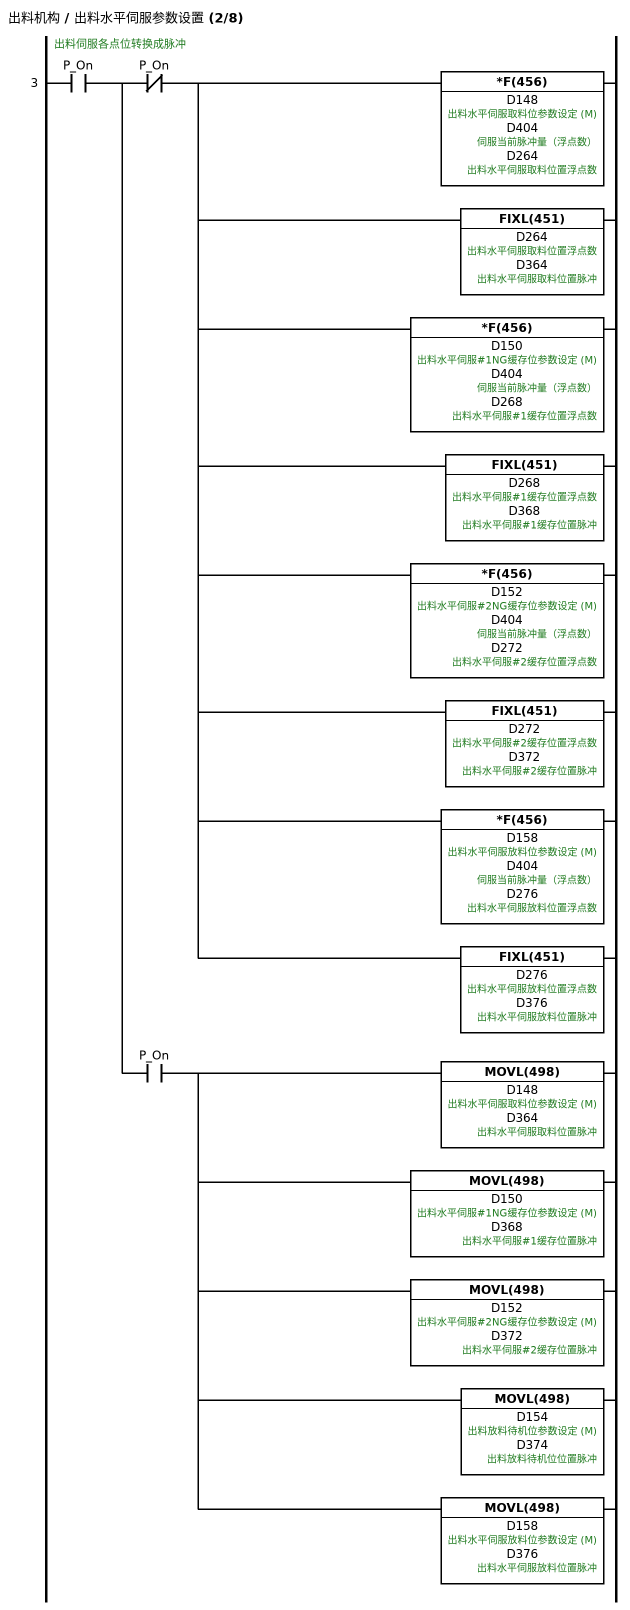
; rung 3: 出料伺服各点位转换成脉冲
LD P_On
OUT TR0
ANDNOT P_On
*F(456) D148 D404 D264  ; 出料水平伺服取料位参数设定 (M), 伺服当前脉冲量（浮点数）, 出料水平伺服取料位置浮点数
FIXL(451) D264 D364  ; 出料水平伺服取料位置浮点数, 出料水平伺服取料位置脉冲
*F(456) D150 D404 D268  ; 出料水平伺服#1NG缓存位参数设定 (M), 伺服当前脉冲量（浮点数）, 出料水平伺服#1缓存位置浮点数
FIXL(451) D268 D368  ; 出料水平伺服#1缓存位置浮点数, 出料水平伺服#1缓存位置脉冲
*F(456) D152 D404 D272  ; 出料水平伺服#2NG缓存位参数设定 (M), 伺服当前脉冲量（浮点数）, 出料水平伺服#2缓存位置浮点数
FIXL(451) D272 D372  ; 出料水平伺服#2缓存位置浮点数, 出料水平伺服#2缓存位置脉冲
*F(456) D158 D404 D276  ; 出料水平伺服放料位参数设定 (M), 伺服当前脉冲量（浮点数）, 出料水平伺服放料位置浮点数
FIXL(451) D276 D376  ; 出料水平伺服放料位置浮点数, 出料水平伺服放料位置脉冲
LD TR0
AND P_On
MOVL(498) D148 D364  ; 出料水平伺服取料位参数设定 (M), 出料水平伺服取料位置脉冲
MOVL(498) D150 D368  ; 出料水平伺服#1NG缓存位参数设定 (M), 出料水平伺服#1缓存位置脉冲
MOVL(498) D152 D372  ; 出料水平伺服#2NG缓存位参数设定 (M), 出料水平伺服#2缓存位置脉冲
MOVL(498) D154 D374  ; 出料放料待机位参数设定 (M), 出料放料待机位位置脉冲
MOVL(498) D158 D376  ; 出料水平伺服放料位参数设定 (M), 出料水平伺服放料位置脉冲

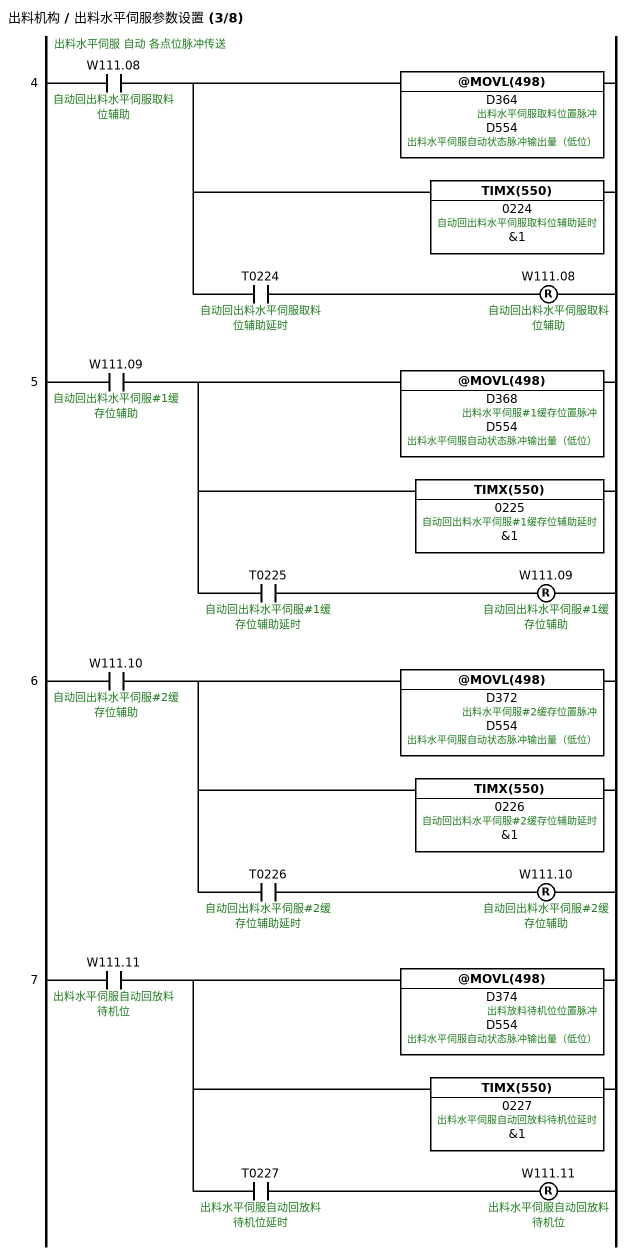
; rung 4: 出料水平伺服 自动 各点位脉冲传送
LD W111.08  ; 自动回出料水平伺服取料位辅助
@MOVL(498) D364 D554  ; 出料水平伺服取料位置脉冲, 出料水平伺服自动状态脉冲输出量（低位）
TIMX(550) 0224 &1  ; 自动回出料水平伺服取料位辅助延时
AND T0224  ; 自动回出料水平伺服取料位辅助延时
RSET W111.08  ; 自动回出料水平伺服取料位辅助
; rung 5
LD W111.09  ; 自动回出料水平伺服#1缓存位辅助
@MOVL(498) D368 D554  ; 出料水平伺服#1缓存位置脉冲, 出料水平伺服自动状态脉冲输出量（低位）
TIMX(550) 0225 &1  ; 自动回出料水平伺服#1缓存位辅助延时
AND T0225  ; 自动回出料水平伺服#1缓存位辅助延时
RSET W111.09  ; 自动回出料水平伺服#1缓存位辅助
; rung 6
LD W111.10  ; 自动回出料水平伺服#2缓存位辅助
@MOVL(498) D372 D554  ; 出料水平伺服#2缓存位置脉冲, 出料水平伺服自动状态脉冲输出量（低位）
TIMX(550) 0226 &1  ; 自动回出料水平伺服#2缓存位辅助延时
AND T0226  ; 自动回出料水平伺服#2缓存位辅助延时
RSET W111.10  ; 自动回出料水平伺服#2缓存位辅助
; rung 7
LD W111.11  ; 出料水平伺服自动回放料待机位
@MOVL(498) D374 D554  ; 出料放料待机位位置脉冲, 出料水平伺服自动状态脉冲输出量（低位）
TIMX(550) 0227 &1  ; 出料水平伺服自动回放料待机位延时
AND T0227  ; 出料水平伺服自动回放料待机位延时
RSET W111.11  ; 出料水平伺服自动回放料待机位

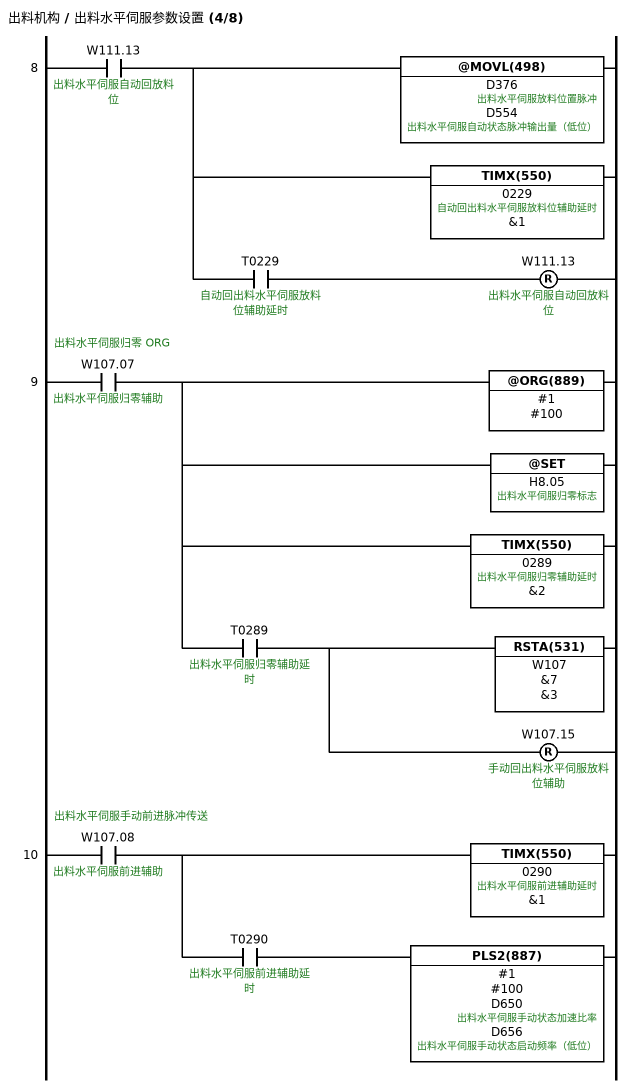
; rung 8
LD W111.13  ; 出料水平伺服自动回放料位
@MOVL(498) D376 D554  ; 出料水平伺服放料位置脉冲, 出料水平伺服自动状态脉冲输出量（低位）
TIMX(550) 0229 &1  ; 自动回出料水平伺服放料位辅助延时
AND T0229  ; 自动回出料水平伺服放料位辅助延时
RSET W111.13  ; 出料水平伺服自动回放料位
; rung 9: 出料水平伺服归零 ORG
LD W107.07  ; 出料水平伺服归零辅助
@ORG(889) #1 #100
@SET H8.05  ; 出料水平伺服归零标志
TIMX(550) 0289 &2  ; 出料水平伺服归零辅助延时
AND T0289  ; 出料水平伺服归零辅助延时
RSTA(531) W107 &7 &3
RSET W107.15  ; 手动回出料水平伺服放料位辅助
; rung 10: 出料水平伺服手动前进脉冲传送
LD W107.08  ; 出料水平伺服前进辅助
TIMX(550) 0290 &1  ; 出料水平伺服前进辅助延时
AND T0290  ; 出料水平伺服前进辅助延时
PLS2(887) #1 #100 D650 D656  ; 出料水平伺服手动状态加速比率, 出料水平伺服手动状态启动频率（低位）

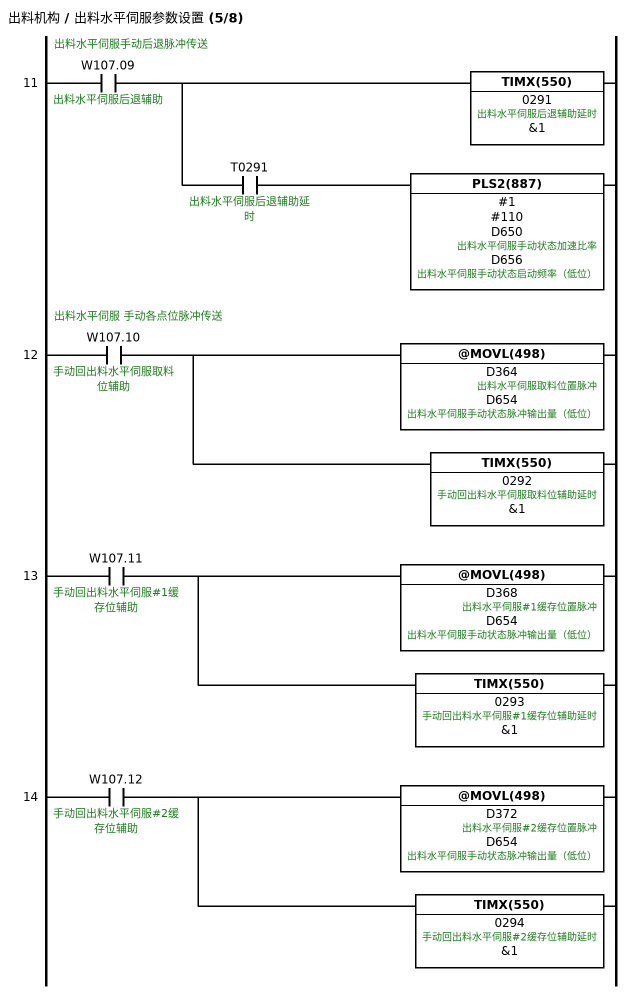
; rung 11: 出料水平伺服手动后退脉冲传送
LD W107.09  ; 出料水平伺服后退辅助
TIMX(550) 0291 &1  ; 出料水平伺服后退辅助延时
AND T0291  ; 出料水平伺服后退辅助延时
PLS2(887) #1 #110 D650 D656  ; 出料水平伺服手动状态加速比率, 出料水平伺服手动状态启动频率（低位）
; rung 12: 出料水平伺服 手动各点位脉冲传送
LD W107.10  ; 手动回出料水平伺服取料位辅助
@MOVL(498) D364 D654  ; 出料水平伺服取料位置脉冲, 出料水平伺服手动状态脉冲输出量（低位）
TIMX(550) 0292 &1  ; 手动回出料水平伺服取料位辅助延时
; rung 13
LD W107.11  ; 手动回出料水平伺服#1缓存位辅助
@MOVL(498) D368 D654  ; 出料水平伺服#1缓存位置脉冲, 出料水平伺服手动状态脉冲输出量（低位）
TIMX(550) 0293 &1  ; 手动回出料水平伺服#1缓存位辅助延时
; rung 14
LD W107.12  ; 手动回出料水平伺服#2缓存位辅助
@MOVL(498) D372 D654  ; 出料水平伺服#2缓存位置脉冲, 出料水平伺服手动状态脉冲输出量（低位）
TIMX(550) 0294 &1  ; 手动回出料水平伺服#2缓存位辅助延时

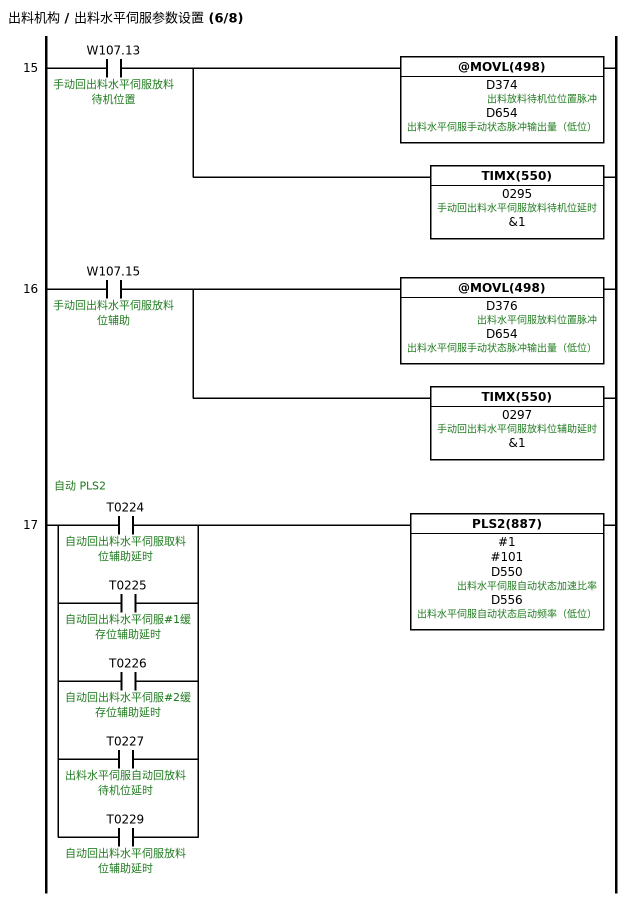
; rung 15
LD W107.13  ; 手动回出料水平伺服放料待机位置
@MOVL(498) D374 D654  ; 出料放料待机位位置脉冲, 出料水平伺服手动状态脉冲输出量（低位）
TIMX(550) 0295 &1  ; 手动回出料水平伺服放料待机位延时
; rung 16
LD W107.15  ; 手动回出料水平伺服放料位辅助
@MOVL(498) D376 D654  ; 出料水平伺服放料位置脉冲, 出料水平伺服手动状态脉冲输出量（低位）
TIMX(550) 0297 &1  ; 手动回出料水平伺服放料位辅助延时
; rung 17: 自动 PLS2
LD T0224  ; 自动回出料水平伺服取料位辅助延时
OR T0225  ; 自动回出料水平伺服#1缓存位辅助延时
OR T0226  ; 自动回出料水平伺服#2缓存位辅助延时
OR T0227  ; 出料水平伺服自动回放料待机位延时
OR T0229  ; 自动回出料水平伺服放料位辅助延时
PLS2(887) #1 #101 D550 D556  ; 出料水平伺服自动状态加速比率, 出料水平伺服自动状态启动频率（低位）

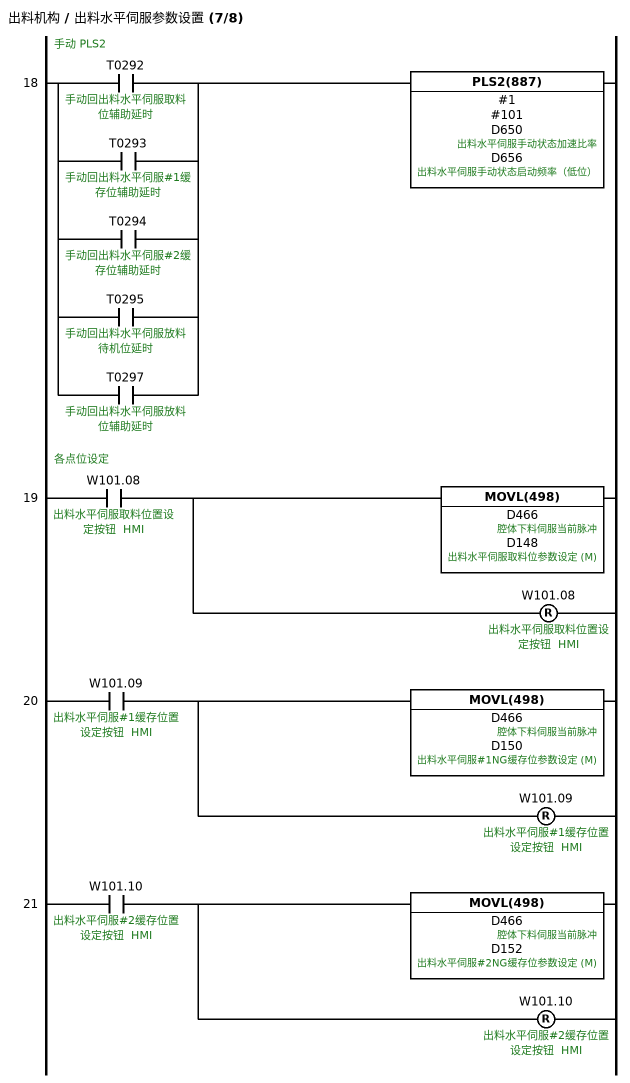
; rung 18: 手动 PLS2
LD T0292  ; 手动回出料水平伺服取料位辅助延时
OR T0293  ; 手动回出料水平伺服#1缓存位辅助延时
OR T0294  ; 手动回出料水平伺服#2缓存位辅助延时
OR T0295  ; 手动回出料水平伺服放料待机位延时
OR T0297  ; 手动回出料水平伺服放料位辅助延时
PLS2(887) #1 #101 D650 D656  ; 出料水平伺服手动状态加速比率, 出料水平伺服手动状态启动频率（低位）
; rung 19: 各点位设定
LD W101.08  ; 出料水平伺服取料位置设定按钮  HMI
MOVL(498) D466 D148  ; 腔体下料伺服当前脉冲, 出料水平伺服取料位参数设定 (M)
RSET W101.08  ; 出料水平伺服取料位置设定按钮  HMI
; rung 20
LD W101.09  ; 出料水平伺服#1缓存位置设定按钮  HMI
MOVL(498) D466 D150  ; 腔体下料伺服当前脉冲, 出料水平伺服#1NG缓存位参数设定 (M)
RSET W101.09  ; 出料水平伺服#1缓存位置设定按钮  HMI
; rung 21
LD W101.10  ; 出料水平伺服#2缓存位置设定按钮  HMI
MOVL(498) D466 D152  ; 腔体下料伺服当前脉冲, 出料水平伺服#2NG缓存位参数设定 (M)
RSET W101.10  ; 出料水平伺服#2缓存位置设定按钮  HMI

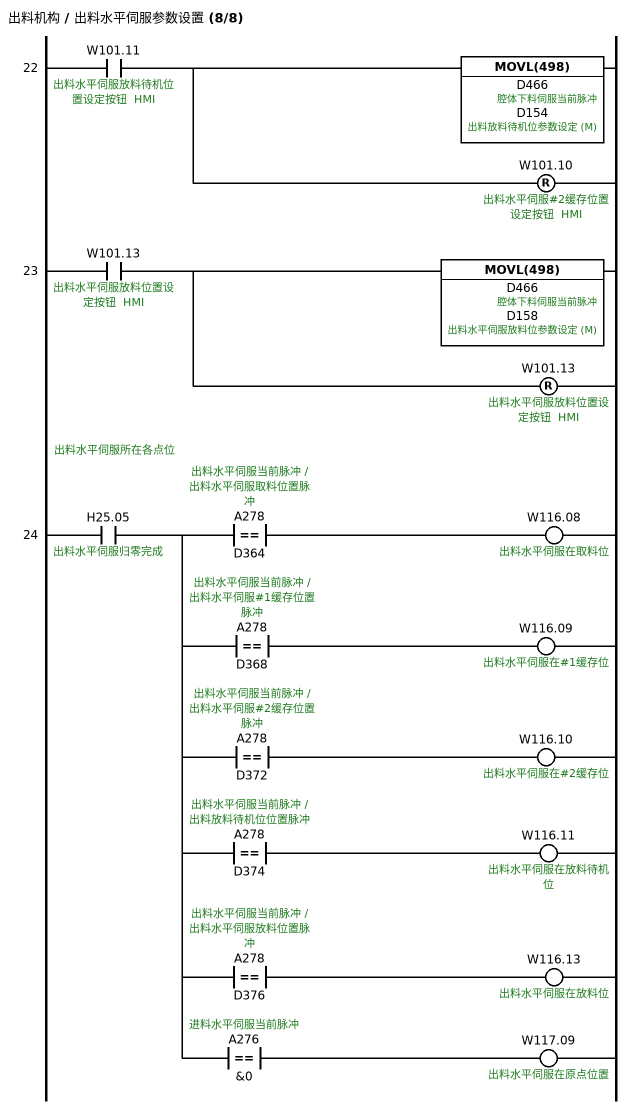
; rung 22
LD W101.11  ; 出料水平伺服放料待机位置设定按钮  HMI
MOVL(498) D466 D154  ; 腔体下料伺服当前脉冲, 出料放料待机位参数设定 (M)
RSET W101.10  ; 出料水平伺服#2缓存位置设定按钮  HMI
; rung 23
LD W101.13  ; 出料水平伺服放料位置设定按钮  HMI
MOVL(498) D466 D158  ; 腔体下料伺服当前脉冲, 出料水平伺服放料位参数设定 (M)
RSET W101.13  ; 出料水平伺服放料位置设定按钮  HMI
; rung 24: 出料水平伺服所在各点位
LD H25.05  ; 出料水平伺服归零完成
OUT TR0
AND=SL(303) A278 D364  ; 出料水平伺服当前脉冲, 出料水平伺服取料位置脉冲
OUT W116.08  ; 出料水平伺服在取料位
LD TR0
AND=SL(303) A278 D368  ; 出料水平伺服当前脉冲, 出料水平伺服#1缓存位置脉冲
OUT W116.09  ; 出料水平伺服在#1缓存位
LD TR0
AND=SL(303) A278 D372  ; 出料水平伺服当前脉冲, 出料水平伺服#2缓存位置脉冲
OUT W116.10  ; 出料水平伺服在#2缓存位
LD TR0
AND=SL(303) A278 D374  ; 出料水平伺服当前脉冲, 出料放料待机位位置脉冲
OUT W116.11  ; 出料水平伺服在放料待机位
LD TR0
AND=SL(303) A278 D376  ; 出料水平伺服当前脉冲, 出料水平伺服放料位置脉冲
OUT W116.13  ; 出料水平伺服在放料位
LD TR0
AND=SL(303) A276 &0  ; 进料水平伺服当前脉冲
OUT W117.09  ; 出料水平伺服在原点位置

### Section 出料升降伺服参数设置

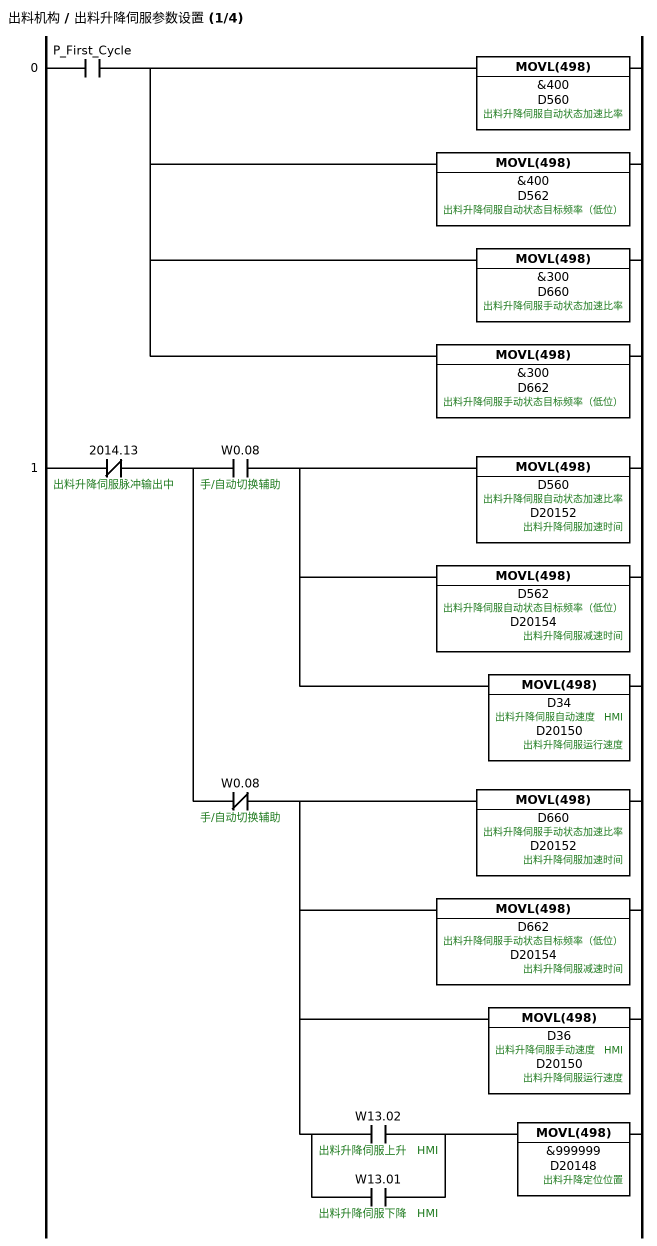
; rung 0
LD P_First_Cycle
MOVL(498) &400 D560  ; 出料升降伺服自动状态加速比率
MOVL(498) &400 D562  ; 出料升降伺服自动状态目标频率（低位）
MOVL(498) &300 D660  ; 出料升降伺服手动状态加速比率
MOVL(498) &300 D662  ; 出料升降伺服手动状态目标频率（低位）
; rung 1
LDNOT 2014.13  ; 出料升降伺服脉冲输出中
OUT TR0
AND W0.08  ; 手/自动切换辅助
MOVL(498) D560 D20152  ; 出料升降伺服自动状态加速比率, 出料升降伺服加速时间
MOVL(498) D562 D20154  ; 出料升降伺服自动状态目标频率（低位）, 出料升降伺服减速时间
MOVL(498) D34 D20150  ; 出料升降伺服自动速度   HMI, 出料升降伺服运行速度
LD TR0
ANDNOT W0.08  ; 手/自动切换辅助
MOVL(498) D660 D20152  ; 出料升降伺服手动状态加速比率, 出料升降伺服加速时间
MOVL(498) D662 D20154  ; 出料升降伺服手动状态目标频率（低位）, 出料升降伺服减速时间
MOVL(498) D36 D20150  ; 出料升降伺服手动速度   HMI, 出料升降伺服运行速度
LD W13.02  ; 出料升降伺服上升   HMI
OR W13.01  ; 出料升降伺服下降   HMI
ANDLD
MOVL(498) &999999 D20148  ; 出料升降定位位置

